PROGRAM MAIN
VAR
END_VAR

P_ModbusRTU_Master();
P_ModbusRTU_Slave();

END_PROGRAM

(* stored: Version 1.1.0.1, ProductVersion 3.1.4024.6
   POU MAIN: Id {3ce17852-111c-47f6-ac91-e7663c6b8f51}, SpecialFunc None *)
